{attribute 'GeneratedUsingTerminal: IODEVICETYPE_ETHERCATPROT'}
{attribute addProperty BoxType "IODEVICETYPE_ETHERCATPROT"}
{attribute addProperty Id "EK1200EK1200_319FD71D204SyncUnitsSyncUnits_67D36DDA18InputsInputs_A65FACA410OutputsOutputs_23C0ED1D6InfoDataInfoData_84133AC922"}
{attribute addProperty CRC "2282533049"}
{attribute addProperty Size "260"}
{attribute addProperty Name "EC1"}
TYPE EC1_880CB0B9 EXTENDS TcoIo.EtcMasterBase_62654B43 :
STRUCT
	{attribute addProperty Name " (EK1200)"}
	{attribute addProperty PreviousPort "EC1 : Master"}
	{attribute addProperty SyncUnit "default"}
	EK1200 : EK1200_319FD71D;
	{attribute addProperty Name "SyncUnits"}
	SyncUnits : SyncUnits_67D36DDA;
	{attribute addProperty Name "Inputs"}
	Inputs : TcoIo.Inputs_A65FACA4;
	{attribute addProperty Name "Outputs"}
	Outputs : TcoIo.Outputs_23C0ED1D;
	{attribute addProperty Name "InfoData"}
	InfoData : TcoIo.InfoData_84133AC9;
END_STRUCT
END_TYPE

(* stored: Version 1.2.0.0
   DUT EC1_880CB0B9: Id {654f8d88-a6f6-411a-a975-e91291d052cc} *)
